// TIA Portal V21 export
DATA_BLOCK "InputValues_DB"   // DB101
{ S7_Optimized_Access := 'TRUE'; DB_Accessible_From_OPC_UA := 'FALSE' }
// stored: AutoNumber false, DBAccessibleFromOPCUA false, DBAccessibleFromWebserver false, MemoryReserve 100
   VAR
      InputsDigital { ExternalWritable := 'False'} : Struct
         EmergencyStop { ExternalAccessible := 'False'; ExternalVisible := 'False'} : Bool;
         Start : Bool;
         Stop : Bool;
         Reset : Bool;
         ContactorON : Array[1..2] of Bool;
         SoftstartON : Array[1..2] of Bool;
         SoftstartBypassed : Array[1..2] of Bool;
         SoftstartFault : Array[1..2] of Bool;
         Protection : Array[1..2] of Bool;
      END_STRUCT;
      TankLevel { ExternalWritable := 'False'} : Array[1..2] of Real;
   END_VAR
BEGIN
END_DATA_BLOCK
